# EPICS autosave request: iocBoot/iocdrvMegamp/as/req/asMenu.req
file configMenu.req P=$(P),CONFIG=$(CONFIG)
file configMenu_settings.req P=$(P),CONFIG=$(CONFIG)
file ioc_settings.req
